(* Schneider Machine Expert - Basic project contoh 1, file version 1.7.0.0 *)
(* ProjectInformations: Name=New project *)

HARDWARE
  Cpu 0: TM221M16R/G
  EthernetConfiguration: NetworkName=M221, IpAllocationMode=FixedAddress, IpAddress=0.0.0.0, SubnetMask=0.0.0.0
  SerialLineConfiguration: Baud=Baud19200, Parity=ParityEven, DataBits=DataBits8, StopBits=StopBits1, PhysicalMedium=PhysicalMediumRs485, TransmissionMode=TransmissionModeModbusRtu, SlaveId=1, Addressing=SlaveAddressing
  MastTask: UsePeriodScanMode=false, PeriodScan=100
  FastTask: Period=255
  CpuBehavior: StartingMode=StartAsPreviousState, AutoSaveRamOnEeprom=true, WatchdogPeriod=250

SYMBOLS  (address, symbol, comment, settings)

POU New POU
  (* SectionNumber=1 *)

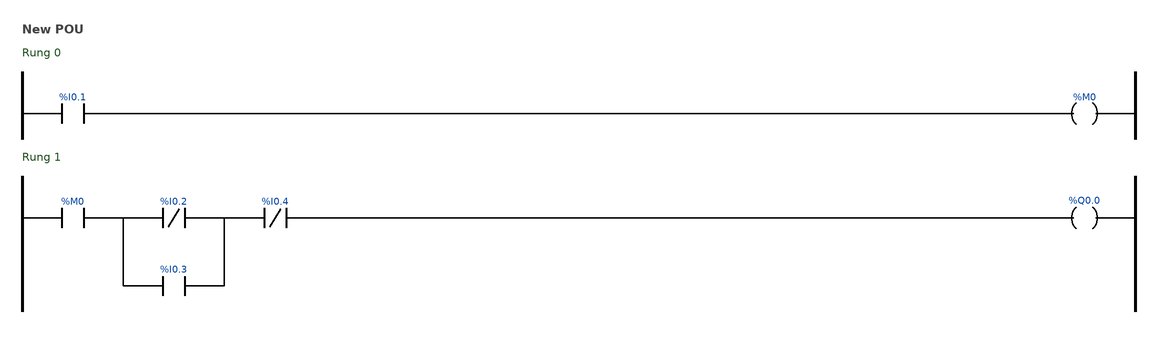

// Rung 0
  LD %I0.1
  ST %M0
  // as ST:
  //   %M0 := %I0.1;

// Rung 1
  LD %M0
  AND(N %I0.2
  OR %I0.3
  )
  ANDN %I0.4
  ST %Q0.0
  // as ST:
  //   %Q0.0 := %M0 AND (NOT %I0.2 OR %I0.3) AND NOT %I0.4;

// Rung 2
  (* no IL stored for this rung *)
